SUBAPPLICATION OPC_PUB_1_FixID_Bool (* Subapplication Type *)
  (* Standard: 61499-2 *)
  (* Version 1.0, 2022-03-09, Maximilian Scharf *)
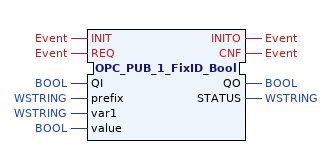
  EVENT_INPUT
    INIT;
    REQ;
  END_EVENT
  EVENT_OUTPUT
    INITO;
    CNF;
  END_EVENT
  VAR_INPUT
    QI : BOOL;
    prefix : WSTRING;
    var1 : WSTRING := STRING#'a';
    value : BOOL;
  END_VAR
  VAR_OUTPUT
    QO : BOOL;
    STATUS : WSTRING;
  END_VAR
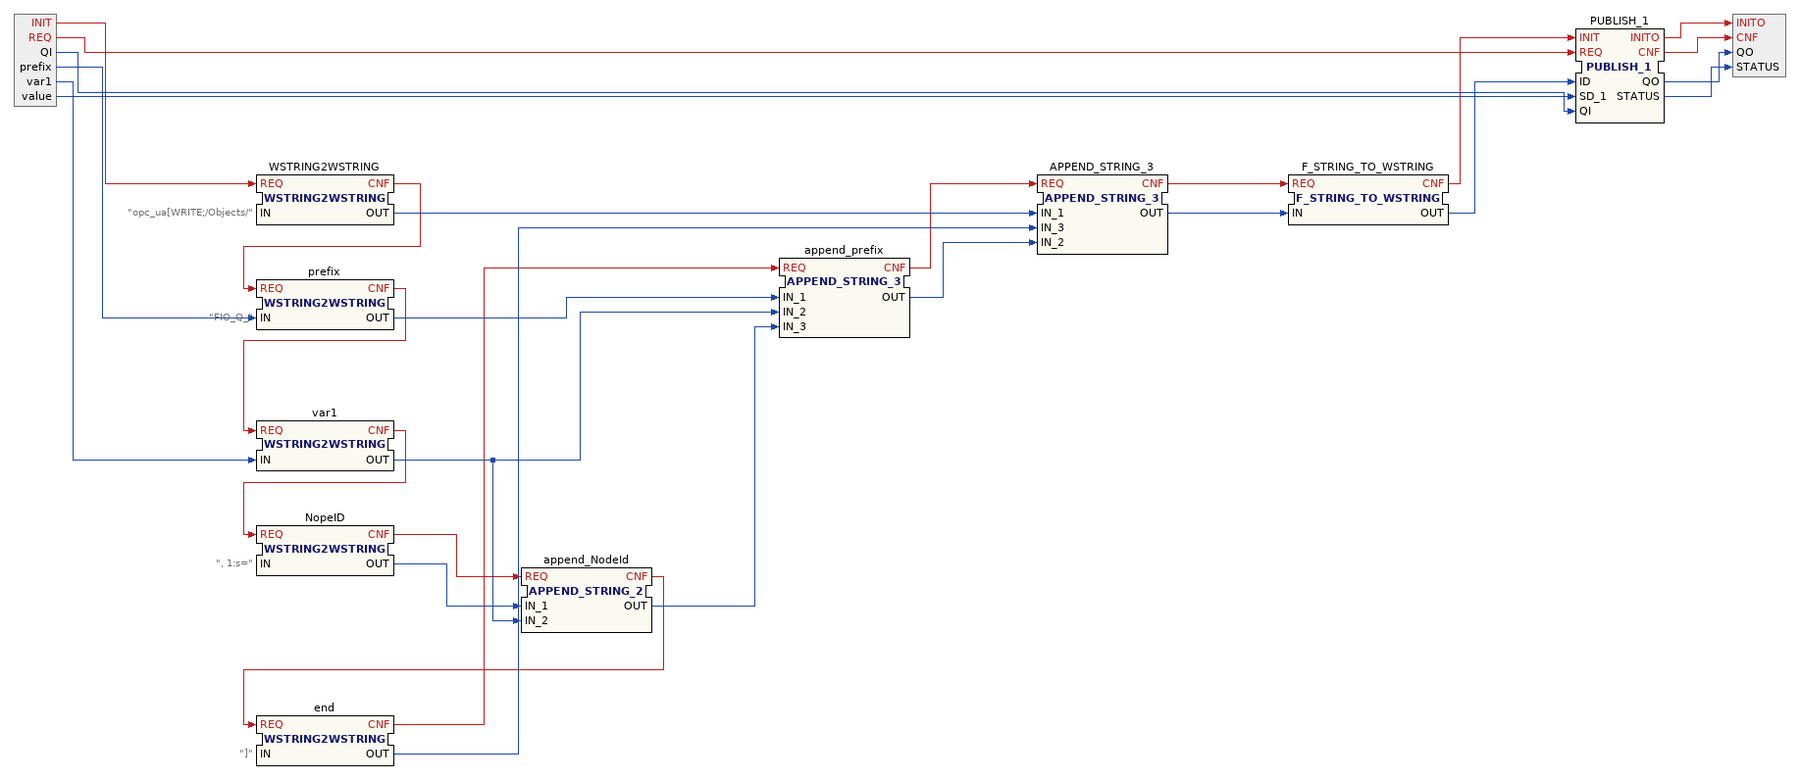
  FBS
    WSTRING2WSTRING : WSTRING2WSTRING(IN := "opc_ua[WRITE;/Objects/");
    F_STRING_TO_WSTRING : F_STRING_TO_WSTRING;
    APPEND_STRING_3 : APPEND_STRING_3;
    end : WSTRING2WSTRING(IN := "]");
    PUBLISH_1 : PUBLISH_1;
    var1 : WSTRING2WSTRING;
    prefix : WSTRING2WSTRING(IN := "FIO_Q_");
    append_prefix : APPEND_STRING_3;
    NopeID : WSTRING2WSTRING(IN := ", 1:s=");
    append_NodeId : APPEND_STRING_2;
  END_FBS
  EVENT_CONNECTIONS
    APPEND_STRING_3.CNF TO F_STRING_TO_WSTRING.REQ;
    F_STRING_TO_WSTRING.CNF TO PUBLISH_1.INIT;
    REQ TO PUBLISH_1.REQ;
    PUBLISH_1.INITO TO INITO;
    PUBLISH_1.CNF TO CNF;
    INIT TO WSTRING2WSTRING.REQ;
    append_prefix.CNF TO APPEND_STRING_3.REQ;
    var1.CNF TO NopeID.REQ;
    WSTRING2WSTRING.CNF TO prefix.REQ;
    prefix.CNF TO var1.REQ;
    append_NodeId.CNF TO end.REQ;
    end.CNF TO append_prefix.REQ;
    NopeID.CNF TO append_NodeId.REQ;
  END_CONNECTIONS
  DATA_CONNECTIONS
    WSTRING2WSTRING.OUT TO APPEND_STRING_3.IN_1;
    APPEND_STRING_3.OUT TO F_STRING_TO_WSTRING.IN;
    F_STRING_TO_WSTRING.OUT TO PUBLISH_1.ID;
    end.OUT TO APPEND_STRING_3.IN_3;
    value TO PUBLISH_1.SD_1;
    PUBLISH_1.QO TO QO;
    PUBLISH_1.STATUS TO STATUS;
    QI TO PUBLISH_1.QI;
    var1 TO var1.IN;
    prefix TO prefix.IN;
    prefix.OUT TO append_prefix.IN_1;
    append_prefix.OUT TO APPEND_STRING_3.IN_2;
    var1.OUT TO append_prefix.IN_2;
    append_NodeId.OUT TO append_prefix.IN_3;
    NopeID.OUT TO append_NodeId.IN_1;
    var1.OUT TO append_NodeId.IN_2;
  END_CONNECTIONS
END_SUBAPPLICATION
